// TwinCAT 3 PLC project sample_delivery
// ProgramVersion: 3.1.4023.0
// libraries:
//   lcls-twincat-sample-delivery, * (SLAC)
//   Tc2_Standard, * (Beckhoff Automation GmbH)
//   Tc2_System, * (Beckhoff Automation GmbH)
//   Tc3_Module, * (Beckhoff Automation GmbH)
// project tree:
//   GVLs/ GVL_SDS.TcGVL
//   / PlcTask.TcTTO, SerialComm.TcTTO
//   POUs/ MAIN.TcPOU, SerialTxRx.TcPOU (not stored)
// real-time tasks:
//   TASK PlcTask: cycle T#10ms, priority 20, ADS port 350
//   TASK SerialComm: cycle T#10ms, priority 1, ADS port 351
// I/O:
//   DEVICE Device 1 (EtherCAT), AmsNetId 172.21.38.25.2.1
//     Term 1 (EK1200)
//     Box 17 (EP9128-0021) [EP9128-0021 8x EtherCAT junction]
//       Term 18 (EP9128-1021) [EP9128-1021 8x EtherCAT junction - Dev A]
//         Box 20 (EP9128-0021)
//       Term 24 (EP9128-2021) [EP9128-2021 8x EtherCAT junction - Dev B]
//     ALI (EP1111) [EP1111-0000 ID-Switch]
//     ALI_X (EP7041-0002)
//     ALI_Y (EP7041-0002)
//     ALI_Z (EP7041-0002)
//     ALI_X_ENC (EP5101-0011)
//     ALI_Gauges (EP3174-0002)
//     ALI_PropValve (EP7041-0002)
//     ALI_Y_ENC (EP5101-0011)
//     ALI_DIO (EP2338-0001)
//     M3 Selector A (EP1111)
//     M3 Selector A Digital IO (EP2338-1001)
//     M3 Selector A Serial IO (EP6002-0002)
//     M3 Selector B (EP1111)
//     M3 Selector B Digital IO (EP2338-1001)
//     M3 Selector B Serial IO (EP6002-0002)
//     PCM A (EP1111) [EP1111-0000 ID-Switch]
//     PCM A (EP4374-0002)
//     PCM A (EP3174-0002)
//     PCM A (EP6002-0002)
//     PCM B (EP1111)
//     PCM B (EP4374-0002)
//     PCM B (EP3174-0002)
//     PCM B (EP6002-0002)
//     Gas_Mani (EP1111)
//     Gas_Mani_NeedleValve (EP4374-0002)
//     Gas_Mani_ValveCtrl (EP2338-0001)
//     Gas_Mani_ValveRbk (EP2338-0001)
//     M3 Selector C (EP1111)
//     M3 Selector C Digital IO (EP2338-1001)
//     M3 Selector C Serial IO (EP6002-0002)
//     M3 Selector D (EP1111)
//     M3 Selector D Digital IO (EP2338-1001)
//     M3 Selector D Serial IO (EP6002-0002)
//     PCM C (EP1111)
//     PCM C (EP4374-0002)
//     PCM C (EP3174-0002)
//     PCM C (EP6002-0002)
//     PCM D (EP1111)
//     PCM D (EP4374-0002)
//     PCM D (EP3174-0002)
//     PCM D (EP6002-0002)
//     Bronkhorst MFM A
//     Bronkhorst MFM B
//     Bronkhorst MFM C
//     Bronkhorst MFM D
//     Solenoid Pair A (EP1111)
//     Solenoid Pair A Digital IO (EP2338-0001)
// variable links:
//   sample-delivery Instance <-> Device 1 (EtherCAT)/Bronkhorst MFM B
//     PlcTask Inputs/GVL_SDS.BronkhorstB.stMFM.i_rFlow <-> TxPDO Map/fMeasure
//     PlcTask Outputs/GVL_SDS.BronkhorstB.stMFM.q_rSetpoint <-> RxPDO Map/fSetpoint
//   sample-delivery Instance <-> Device 1 (EtherCAT)/Gas_Mani_ValveCtrl (EP2338-0001)
//     PlcTask Outputs/GVL_SDS.GasMan.stValve[{1..7}].qxDO <-> Channel {9..15}/Output  (7 links)
//   sample-delivery Instance <-> Device 1 (EtherCAT)/Gas_Mani_ValveRbk (EP2338-0001)
//     PlcTask Inputs/GVL_SDS.GasMan.stValve[{1..7}].ixOPN <-> Channel {1..7}/Input  (7 links)
//   sample-delivery Instance <-> Device 1 (EtherCAT)/M3 Selector A Digital IO (EP2338-1001)
//     PlcTask Outputs/GVL_SDS.M3SelectorA.stShaker01.q_xPwrDO <-> Channel 9/Output
//     PlcTask Outputs/GVL_SDS.M3SelectorA.stShaker02.q_xPwrDO <-> Channel 10/Output
//     PlcTask Outputs/GVL_SDS.M3SelectorA.stShaker03.q_xPwrDO <-> Channel 11/Output
//     PlcTask Outputs/GVL_SDS.M3SelectorA.stShaker04.q_xPwrDO <-> Channel 12/Output
//   sample-delivery Instance <-> Device 1 (EtherCAT)/M3 Selector A Serial IO (EP6002-0002)
//     SerialComm Inputs/GVL_SDS.M3SelectorA.stSensSerial.stComIn/Status <-> COM TxPDO-Map Inputs Channel 1/Status
//     SerialComm Inputs/GVL_SDS.M3SelectorA.stViciSerial.stComIn/Status <-> COM TxPDO-Map Inputs Channel 2/Status
//   sample-delivery Instance <-> Device 1 (EtherCAT)/M3 Selector B Digital IO (EP2338-1001)
//     PlcTask Outputs/GVL_SDS.M3SelectorB.stShaker01.q_xPwrDO <-> Channel 9/Output
//     PlcTask Outputs/GVL_SDS.M3SelectorB.stShaker02.q_xPwrDO <-> Channel 10/Output
//     PlcTask Outputs/GVL_SDS.M3SelectorB.stShaker03.q_xPwrDO <-> Channel 11/Output
//     PlcTask Outputs/GVL_SDS.M3SelectorB.stShaker04.q_xPwrDO <-> Channel 12/Output
//   sample-delivery Instance <-> Device 1 (EtherCAT)/M3 Selector B Serial IO (EP6002-0002)
//     SerialComm Inputs/GVL_SDS.M3SelectorB.stSensSerial.stComIn/Status <-> COM TxPDO-Map Inputs Channel 1/Status
//     SerialComm Inputs/GVL_SDS.M3SelectorB.stViciSerial.stComIn/Status <-> COM TxPDO-Map Inputs Channel 2/Status
//   sample-delivery Instance <-> Device 1 (EtherCAT)/M3 Selector C Digital IO (EP2338-1001)
//     PlcTask Outputs/GVL_SDS.M3SelectorC.stShaker01.q_xPwrDO <-> Channel 9/Output
//     PlcTask Outputs/GVL_SDS.M3SelectorC.stShaker02.q_xPwrDO <-> Channel 10/Output
//     PlcTask Outputs/GVL_SDS.M3SelectorC.stShaker03.q_xPwrDO <-> Channel 11/Output
//     PlcTask Outputs/GVL_SDS.M3SelectorC.stShaker04.q_xPwrDO <-> Channel 12/Output
//   sample-delivery Instance <-> Device 1 (EtherCAT)/M3 Selector C Serial IO (EP6002-0002)
//     SerialComm Inputs/GVL_SDS.M3SelectorC.stSensSerial.stComIn/Status <-> COM TxPDO-Map Inputs Channel 1/Status
//     SerialComm Inputs/GVL_SDS.M3SelectorC.stViciSerial.stComIn/Status <-> COM TxPDO-Map Inputs Channel 2/Status
//   sample-delivery Instance <-> Device 1 (EtherCAT)/M3 Selector D Digital IO (EP2338-1001)
//     PlcTask Outputs/GVL_SDS.M3SelectorD.stShaker01.q_xPwrDO <-> Channel 9/Output
//     PlcTask Outputs/GVL_SDS.M3SelectorD.stShaker02.q_xPwrDO <-> Channel 10/Output
//     PlcTask Outputs/GVL_SDS.M3SelectorD.stShaker03.q_xPwrDO <-> Channel 11/Output
//     PlcTask Outputs/GVL_SDS.M3SelectorD.stShaker04.q_xPwrDO <-> Channel 12/Output
//   sample-delivery Instance <-> Device 1 (EtherCAT)/M3 Selector D Serial IO (EP6002-0002)
//     SerialComm Inputs/GVL_SDS.M3SelectorD.stSensSerial.stComIn/Status <-> COM TxPDO-Map Inputs Channel 1/Status
//     SerialComm Inputs/GVL_SDS.M3SelectorD.stViciSerial.stComIn/Status <-> COM TxPDO-Map Inputs Channel 2/Status
//   sample-delivery Instance <-> Device 1 (EtherCAT)/PCM A (EP1111)
//     PlcTask Inputs/GVL_SDS.PCMA.stBaseIO.i_SyncUnitWC <-> WcState/WcState
//   sample-delivery Instance <-> Device 1 (EtherCAT)/PCM A (EP4374-0002)
//     PlcTask Inputs/GVL_SDS.PCMA.stPropAir1.i_iPressRB <-> AI Inputs Channel 1/Value
//     PlcTask Inputs/GVL_SDS.PCMA.stPropAir2.i_iPressRB <-> AI Inputs Channel 2/Value
//     PlcTask Outputs/GVL_SDS.PCMA.stPropAir1.q_iPressCt <-> AO Outputs Channel 3/Analog output
//     PlcTask Outputs/GVL_SDS.PCMA.stPropAir2.q_iPressCt <-> AO Outputs Channel 4/Analog output
//   sample-delivery Instance <-> Device 1 (EtherCAT)/PCM A (EP6002-0002)
//     SerialComm Inputs/GVL_SDS.PCMA.stSerial1.stComIn/D[0] <-> COM TxPDO-Map Inputs Channel 1/Data In 0
//     SerialComm Inputs/GVL_SDS.PCMA.stSerial1.stComIn/D[10] <-> COM TxPDO-Map Inputs Channel 1/Data In 10
//     SerialComm Inputs/GVL_SDS.PCMA.stSerial1.stComIn/D[11] <-> COM TxPDO-Map Inputs Channel 1/Data In 11
//     SerialComm Inputs/GVL_SDS.PCMA.stSerial1.stComIn/D[12] <-> COM TxPDO-Map Inputs Channel 1/Data In 12
//     SerialComm Inputs/GVL_SDS.PCMA.stSerial1.stComIn/D[13] <-> COM TxPDO-Map Inputs Channel 1/Data In 13
//     SerialComm Inputs/GVL_SDS.PCMA.stSerial1.stComIn/D[14] <-> COM TxPDO-Map Inputs Channel 1/Data In 14
//     SerialComm Inputs/GVL_SDS.PCMA.stSerial1.stComIn/D[15] <-> COM TxPDO-Map Inputs Channel 1/Data In 15
//     SerialComm Inputs/GVL_SDS.PCMA.stSerial1.stComIn/D[16] <-> COM TxPDO-Map Inputs Channel 1/Data In 16
//     SerialComm Inputs/GVL_SDS.PCMA.stSerial1.stComIn/D[17] <-> COM TxPDO-Map Inputs Channel 1/Data In 17
//     SerialComm Inputs/GVL_SDS.PCMA.stSerial1.stComIn/D[18] <-> COM TxPDO-Map Inputs Channel 1/Data In 18
//     SerialComm Inputs/GVL_SDS.PCMA.stSerial1.stComIn/D[19] <-> COM TxPDO-Map Inputs Channel 1/Data In 19
//     SerialComm Inputs/GVL_SDS.PCMA.stSerial1.stComIn/D[1] <-> COM TxPDO-Map Inputs Channel 1/Data In 1
//     SerialComm Inputs/GVL_SDS.PCMA.stSerial1.stComIn/D[20] <-> COM TxPDO-Map Inputs Channel 1/Data In 20
//     SerialComm Inputs/GVL_SDS.PCMA.stSerial1.stComIn/D[21] <-> COM TxPDO-Map Inputs Channel 1/Data In 21
//     SerialComm Inputs/GVL_SDS.PCMA.stSerial1.stComIn/D[2] <-> COM TxPDO-Map Inputs Channel 1/Data In 2
//     SerialComm Inputs/GVL_SDS.PCMA.stSerial1.stComIn/D[3] <-> COM TxPDO-Map Inputs Channel 1/Data In 3
//     SerialComm Inputs/GVL_SDS.PCMA.stSerial1.stComIn/D[4] <-> COM TxPDO-Map Inputs Channel 1/Data In 4
//     SerialComm Inputs/GVL_SDS.PCMA.stSerial1.stComIn/D[5] <-> COM TxPDO-Map Inputs Channel 1/Data In 5
//     SerialComm Inputs/GVL_SDS.PCMA.stSerial1.stComIn/D[6] <-> COM TxPDO-Map Inputs Channel 1/Data In 6
//     SerialComm Inputs/GVL_SDS.PCMA.stSerial1.stComIn/D[7] <-> COM TxPDO-Map Inputs Channel 1/Data In 7
//     SerialComm Inputs/GVL_SDS.PCMA.stSerial1.stComIn/D[8] <-> COM TxPDO-Map Inputs Channel 1/Data In 8
//     SerialComm Inputs/GVL_SDS.PCMA.stSerial1.stComIn/D[9] <-> COM TxPDO-Map Inputs Channel 1/Data In 9
//     SerialComm Inputs/GVL_SDS.PCMA.stSerial2.stComIn/D[0] <-> COM TxPDO-Map Inputs Channel 2/Data In 0
//     SerialComm Inputs/GVL_SDS.PCMA.stSerial2.stComIn/D[10] <-> COM TxPDO-Map Inputs Channel 2/Data In 10
//     SerialComm Inputs/GVL_SDS.PCMA.stSerial2.stComIn/D[11] <-> COM TxPDO-Map Inputs Channel 2/Data In 11
//     SerialComm Inputs/GVL_SDS.PCMA.stSerial2.stComIn/D[12] <-> COM TxPDO-Map Inputs Channel 2/Data In 12
//     SerialComm Inputs/GVL_SDS.PCMA.stSerial2.stComIn/D[13] <-> COM TxPDO-Map Inputs Channel 2/Data In 13
//     SerialComm Inputs/GVL_SDS.PCMA.stSerial2.stComIn/D[14] <-> COM TxPDO-Map Inputs Channel 2/Data In 14
//     SerialComm Inputs/GVL_SDS.PCMA.stSerial2.stComIn/D[15] <-> COM TxPDO-Map Inputs Channel 2/Data In 15
//     SerialComm Inputs/GVL_SDS.PCMA.stSerial2.stComIn/D[16] <-> COM TxPDO-Map Inputs Channel 2/Data In 16
//     SerialComm Inputs/GVL_SDS.PCMA.stSerial2.stComIn/D[17] <-> COM TxPDO-Map Inputs Channel 2/Data In 17
//     SerialComm Inputs/GVL_SDS.PCMA.stSerial2.stComIn/D[18] <-> COM TxPDO-Map Inputs Channel 2/Data In 18
//     SerialComm Inputs/GVL_SDS.PCMA.stSerial2.stComIn/D[19] <-> COM TxPDO-Map Inputs Channel 2/Data In 19
//     SerialComm Inputs/GVL_SDS.PCMA.stSerial2.stComIn/D[1] <-> COM TxPDO-Map Inputs Channel 2/Data In 1
//     SerialComm Inputs/GVL_SDS.PCMA.stSerial2.stComIn/D[20] <-> COM TxPDO-Map Inputs Channel 2/Data In 20
//     SerialComm Inputs/GVL_SDS.PCMA.stSerial2.stComIn/D[21] <-> COM TxPDO-Map Inputs Channel 2/Data In 21
//     SerialComm Inputs/GVL_SDS.PCMA.stSerial2.stComIn/D[2] <-> COM TxPDO-Map Inputs Channel 2/Data In 2
//     SerialComm Inputs/GVL_SDS.PCMA.stSerial2.stComIn/D[3] <-> COM TxPDO-Map Inputs Channel 2/Data In 3
//     SerialComm Inputs/GVL_SDS.PCMA.stSerial2.stComIn/D[4] <-> COM TxPDO-Map Inputs Channel 2/Data In 4
//     SerialComm Inputs/GVL_SDS.PCMA.stSerial2.stComIn/D[5] <-> COM TxPDO-Map Inputs Channel 2/Data In 5
//     SerialComm Inputs/GVL_SDS.PCMA.stSerial2.stComIn/D[6] <-> COM TxPDO-Map Inputs Channel 2/Data In 6
//     SerialComm Inputs/GVL_SDS.PCMA.stSerial2.stComIn/D[7] <-> COM TxPDO-Map Inputs Channel 2/Data In 7
//     SerialComm Inputs/GVL_SDS.PCMA.stSerial2.stComIn/D[8] <-> COM TxPDO-Map Inputs Channel 2/Data In 8
//     SerialComm Inputs/GVL_SDS.PCMA.stSerial2.stComIn/D[9] <-> COM TxPDO-Map Inputs Channel 2/Data In 9
//     SerialComm Inputs/GVL_SDS.PCMA.stSerial1.stComIn/Status <-> COM TxPDO-Map Inputs Channel 1/Status
//     SerialComm Inputs/GVL_SDS.PCMA.stSerial2.stComIn/Status <-> COM TxPDO-Map Inputs Channel 2/Status
//     SerialComm Outputs/GVL_SDS.PCMA.stSerial1.stComOut/Ctrl <-> COM RxPDO-Map Outputs Channel 1/Ctrl
//     SerialComm Outputs/GVL_SDS.PCMA.stSerial2.stComOut/Ctrl <-> COM RxPDO-Map Outputs Channel 2/Ctrl
//     SerialComm Outputs/GVL_SDS.PCMA.stSerial1.stComOut/D[0] <-> COM RxPDO-Map Outputs Channel 1/Data Out 0
//     SerialComm Outputs/GVL_SDS.PCMA.stSerial1.stComOut/D[10] <-> COM RxPDO-Map Outputs Channel 1/Data Out 10
//     SerialComm Outputs/GVL_SDS.PCMA.stSerial1.stComOut/D[11] <-> COM RxPDO-Map Outputs Channel 1/Data Out 11
//     SerialComm Outputs/GVL_SDS.PCMA.stSerial1.stComOut/D[12] <-> COM RxPDO-Map Outputs Channel 1/Data Out 12
//     SerialComm Outputs/GVL_SDS.PCMA.stSerial1.stComOut/D[13] <-> COM RxPDO-Map Outputs Channel 1/Data Out 13
//     SerialComm Outputs/GVL_SDS.PCMA.stSerial1.stComOut/D[14] <-> COM RxPDO-Map Outputs Channel 1/Data Out 14
//     SerialComm Outputs/GVL_SDS.PCMA.stSerial1.stComOut/D[15] <-> COM RxPDO-Map Outputs Channel 1/Data Out 15
//     SerialComm Outputs/GVL_SDS.PCMA.stSerial1.stComOut/D[16] <-> COM RxPDO-Map Outputs Channel 1/Data Out 16
//     SerialComm Outputs/GVL_SDS.PCMA.stSerial1.stComOut/D[17] <-> COM RxPDO-Map Outputs Channel 1/Data Out 17
//     SerialComm Outputs/GVL_SDS.PCMA.stSerial1.stComOut/D[18] <-> COM RxPDO-Map Outputs Channel 1/Data Out 18
//     SerialComm Outputs/GVL_SDS.PCMA.stSerial1.stComOut/D[19] <-> COM RxPDO-Map Outputs Channel 1/Data Out 19
//     SerialComm Outputs/GVL_SDS.PCMA.stSerial1.stComOut/D[1] <-> COM RxPDO-Map Outputs Channel 1/Data Out 1
//     SerialComm Outputs/GVL_SDS.PCMA.stSerial1.stComOut/D[20] <-> COM RxPDO-Map Outputs Channel 1/Data Out 20
//     SerialComm Outputs/GVL_SDS.PCMA.stSerial1.stComOut/D[21] <-> COM RxPDO-Map Outputs Channel 1/Data Out 21
//     SerialComm Outputs/GVL_SDS.PCMA.stSerial1.stComOut/D[2] <-> COM RxPDO-Map Outputs Channel 1/Data Out 2
//     SerialComm Outputs/GVL_SDS.PCMA.stSerial1.stComOut/D[3] <-> COM RxPDO-Map Outputs Channel 1/Data Out 3
//     SerialComm Outputs/GVL_SDS.PCMA.stSerial1.stComOut/D[4] <-> COM RxPDO-Map Outputs Channel 1/Data Out 4
//     SerialComm Outputs/GVL_SDS.PCMA.stSerial1.stComOut/D[5] <-> COM RxPDO-Map Outputs Channel 1/Data Out 5
//     SerialComm Outputs/GVL_SDS.PCMA.stSerial1.stComOut/D[6] <-> COM RxPDO-Map Outputs Channel 1/Data Out 6
//     SerialComm Outputs/GVL_SDS.PCMA.stSerial1.stComOut/D[7] <-> COM RxPDO-Map Outputs Channel 1/Data Out 7
//     SerialComm Outputs/GVL_SDS.PCMA.stSerial1.stComOut/D[8] <-> COM RxPDO-Map Outputs Channel 1/Data Out 8
//     SerialComm Outputs/GVL_SDS.PCMA.stSerial1.stComOut/D[9] <-> COM RxPDO-Map Outputs Channel 1/Data Out 9
//     SerialComm Outputs/GVL_SDS.PCMA.stSerial2.stComOut/D[0] <-> COM RxPDO-Map Outputs Channel 2/Data Out 0
//     SerialComm Outputs/GVL_SDS.PCMA.stSerial2.stComOut/D[10] <-> COM RxPDO-Map Outputs Channel 2/Data Out 10
//     SerialComm Outputs/GVL_SDS.PCMA.stSerial2.stComOut/D[11] <-> COM RxPDO-Map Outputs Channel 2/Data Out 11
//     SerialComm Outputs/GVL_SDS.PCMA.stSerial2.stComOut/D[12] <-> COM RxPDO-Map Outputs Channel 2/Data Out 12
//     SerialComm Outputs/GVL_SDS.PCMA.stSerial2.stComOut/D[13] <-> COM RxPDO-Map Outputs Channel 2/Data Out 13
//     SerialComm Outputs/GVL_SDS.PCMA.stSerial2.stComOut/D[14] <-> COM RxPDO-Map Outputs Channel 2/Data Out 14
//     SerialComm Outputs/GVL_SDS.PCMA.stSerial2.stComOut/D[15] <-> COM RxPDO-Map Outputs Channel 2/Data Out 15
//     SerialComm Outputs/GVL_SDS.PCMA.stSerial2.stComOut/D[16] <-> COM RxPDO-Map Outputs Channel 2/Data Out 16
//     SerialComm Outputs/GVL_SDS.PCMA.stSerial2.stComOut/D[17] <-> COM RxPDO-Map Outputs Channel 2/Data Out 17
//     SerialComm Outputs/GVL_SDS.PCMA.stSerial2.stComOut/D[18] <-> COM RxPDO-Map Outputs Channel 2/Data Out 18
//     SerialComm Outputs/GVL_SDS.PCMA.stSerial2.stComOut/D[19] <-> COM RxPDO-Map Outputs Channel 2/Data Out 19
//     SerialComm Outputs/GVL_SDS.PCMA.stSerial2.stComOut/D[1] <-> COM RxPDO-Map Outputs Channel 2/Data Out 1
//     SerialComm Outputs/GVL_SDS.PCMA.stSerial2.stComOut/D[20] <-> COM RxPDO-Map Outputs Channel 2/Data Out 20
//     SerialComm Outputs/GVL_SDS.PCMA.stSerial2.stComOut/D[21] <-> COM RxPDO-Map Outputs Channel 2/Data Out 21
//     SerialComm Outputs/GVL_SDS.PCMA.stSerial2.stComOut/D[2] <-> COM RxPDO-Map Outputs Channel 2/Data Out 2
//     SerialComm Outputs/GVL_SDS.PCMA.stSerial2.stComOut/D[3] <-> COM RxPDO-Map Outputs Channel 2/Data Out 3
//     SerialComm Outputs/GVL_SDS.PCMA.stSerial2.stComOut/D[4] <-> COM RxPDO-Map Outputs Channel 2/Data Out 4
//     SerialComm Outputs/GVL_SDS.PCMA.stSerial2.stComOut/D[5] <-> COM RxPDO-Map Outputs Channel 2/Data Out 5
//     SerialComm Outputs/GVL_SDS.PCMA.stSerial2.stComOut/D[6] <-> COM RxPDO-Map Outputs Channel 2/Data Out 6
//     SerialComm Outputs/GVL_SDS.PCMA.stSerial2.stComOut/D[7] <-> COM RxPDO-Map Outputs Channel 2/Data Out 7
//     SerialComm Outputs/GVL_SDS.PCMA.stSerial2.stComOut/D[8] <-> COM RxPDO-Map Outputs Channel 2/Data Out 8
//     SerialComm Outputs/GVL_SDS.PCMA.stSerial2.stComOut/D[9] <-> COM RxPDO-Map Outputs Channel 2/Data Out 9
//   sample-delivery Instance <-> Device 1 (EtherCAT)/PCM B (EP1111)
//     PlcTask Inputs/GVL_SDS.PCMB.stBaseIO.i_SyncUnitWC <-> WcState/WcState
//   sample-delivery Instance <-> Device 1 (EtherCAT)/PCM B (EP4374-0002)
//     PlcTask Inputs/GVL_SDS.PCMB.stPropAir1.i_iPressRB <-> AI Inputs Channel 1/Value
//     PlcTask Inputs/GVL_SDS.PCMB.stPropAir2.i_iPressRB <-> AI Inputs Channel 2/Value
//     PlcTask Outputs/GVL_SDS.PCMB.stPropAir1.q_iPressCt <-> AO Outputs Channel 3/Analog output
//     PlcTask Outputs/GVL_SDS.PCMB.stPropAir2.q_iPressCt <-> AO Outputs Channel 4/Analog output
//   sample-delivery Instance <-> Device 1 (EtherCAT)/PCM B (EP6002-0002)
//     SerialComm Inputs/GVL_SDS.PCMB.stSerial1.stComIn/Status <-> COM TxPDO-Map Inputs Channel 1/Status
//     SerialComm Inputs/GVL_SDS.PCMB.stSerial2.stComIn/Status <-> COM TxPDO-Map Inputs Channel 2/Status
//     SerialComm Outputs/GVL_SDS.PCMB.stSerial1.stComOut/Ctrl <-> COM RxPDO-Map Outputs Channel 1/Ctrl
//     SerialComm Outputs/GVL_SDS.PCMB.stSerial2.stComOut/Ctrl <-> COM RxPDO-Map Outputs Channel 2/Ctrl
//   sample-delivery Instance <-> Device 1 (EtherCAT)/PCM C (EP1111)
//     PlcTask Inputs/GVL_SDS.PCMC.stBaseIO.i_SyncUnitWC <-> WcState/WcState
//   sample-delivery Instance <-> Device 1 (EtherCAT)/PCM C (EP4374-0002)
//     PlcTask Inputs/GVL_SDS.PCMC.stPropAir1.i_iPressRB <-> AI Inputs Channel 1/Value
//     PlcTask Inputs/GVL_SDS.PCMC.stPropAir2.i_iPressRB <-> AI Inputs Channel 2/Value
//     PlcTask Outputs/GVL_SDS.PCMC.stPropAir1.q_iPressCt <-> AO Outputs Channel 3/Analog output
//     PlcTask Outputs/GVL_SDS.PCMC.stPropAir2.q_iPressCt <-> AO Outputs Channel 4/Analog output
//   sample-delivery Instance <-> Device 1 (EtherCAT)/PCM C (EP6002-0002)
//     SerialComm Inputs/GVL_SDS.PCMC.stSerial1.stComIn/Status <-> COM TxPDO-Map Inputs Channel 1/Status
//     SerialComm Inputs/GVL_SDS.PCMC.stSerial2.stComIn/Status <-> COM TxPDO-Map Inputs Channel 2/Status
//     SerialComm Outputs/GVL_SDS.PCMC.stSerial1.stComOut/Ctrl <-> COM RxPDO-Map Outputs Channel 1/Ctrl
//     SerialComm Outputs/GVL_SDS.PCMC.stSerial2.stComOut/Ctrl <-> COM RxPDO-Map Outputs Channel 2/Ctrl
//   sample-delivery Instance <-> Device 1 (EtherCAT)/PCM D (EP1111)
//     PlcTask Inputs/GVL_SDS.PCMD.stBaseIO.i_SyncUnitWC <-> WcState/WcState
//   sample-delivery Instance <-> Device 1 (EtherCAT)/PCM D (EP4374-0002)
//     PlcTask Inputs/GVL_SDS.PCMD.stPropAir1.i_iPressRB <-> AI Inputs Channel 1/Value
//     PlcTask Inputs/GVL_SDS.PCMD.stPropAir2.i_iPressRB <-> AI Inputs Channel 2/Value
//     PlcTask Outputs/GVL_SDS.PCMD.stPropAir1.q_iPressCt <-> AO Outputs Channel 3/Analog output
//     PlcTask Outputs/GVL_SDS.PCMD.stPropAir2.q_iPressCt <-> AO Outputs Channel 4/Analog output
//   sample-delivery Instance <-> Device 1 (EtherCAT)/PCM D (EP6002-0002)
//     SerialComm Inputs/GVL_SDS.PCMD.stSerial1.stComIn/Status <-> COM TxPDO-Map Inputs Channel 1/Status
//     SerialComm Inputs/GVL_SDS.PCMD.stSerial2.stComIn/Status <-> COM TxPDO-Map Inputs Channel 2/Status
//     SerialComm Outputs/GVL_SDS.PCMD.stSerial1.stComOut/Ctrl <-> COM RxPDO-Map Outputs Channel 1/Ctrl
//     SerialComm Outputs/GVL_SDS.PCMD.stSerial2.stComOut/Ctrl <-> COM RxPDO-Map Outputs Channel 2/Ctrl
//   sample-delivery Instance <-> Device 1 (EtherCAT)/Solenoid Pair A Digital IO (EP2338-0001)
//     PlcTask Outputs/GVL_SDS.SolenoidPairA.q_xDO1 <-> Channel 9/Output
//     PlcTask Outputs/GVL_SDS.SolenoidPairA.q_xDO2 <-> Channel 10/Output

CONFIGURATION sample_delivery
    RESOURCE PLC ON TwinCAT3
        TASK PlcTask(INTERVAL := T#10ms, PRIORITY := 20);
        TASK SerialComm(INTERVAL := T#10ms, PRIORITY := 1);
        PROGRAM MAIN WITH PlcTask : MAIN;
        PROGRAM SerialTxRx WITH SerialComm : SerialTxRx;
    END_RESOURCE
END_CONFIGURATION

// ---- GVLs/GVL_SDS.TcGVL
VAR_GLOBAL
	
// TODO: FIX Linking for Devices will be deployed
//  Working: Bronkhorst MFM B
{attribute 'pytmc' := 'pv: XCS:SDS:SEL:A'}
{attribute 'TcLinkTo' := '.stSensSerial.stComIn.Status := TIIB[M3 Selector A Serial IO (EP6002-0002)]^COM TxPDO-Map Inputs Channel 1^Status;
                          .stViciSerial.stComIn.Status := TIIB[M3 Selector A Serial IO (EP6002-0002)]^COM TxPDO-Map Inputs Channel 2^Status;
                          .stSensSerial.stComOut.Ctrl := TIID^MAIN (EtherCAT)^M3 Selector A Serial IO (EP6002-0002)^COM RxPDO-Map Outputs Channel 1^Ctrl;
                          .stViciSerial.stComOut.Ctrl := TIID^MAIN (EtherCAT)^M3 Selector A Serial IO (EP6002-0002)^COM RxPDO-Map Outputs Channel 2^Ctrl;
                          .stShaker01.q_xPwrDO := TIIB[M3 Selector A Digital IO (EP2338-1001)]^Channel 9^Output;
                          .stShaker02.q_xPwrDO := TIIB[M3 Selector A Digital IO (EP2338-1001)]^Channel 10^Output;
                          .stShaker03.q_xPwrDO := TIIB[M3 Selector A Digital IO (EP2338-1001)]^Channel 11^Output;
                          .stShaker04.q_xPwrDO := TIIB[M3 Selector A Digital IO (EP2338-1001)]^Channel 12^Output;
                          .stBaseIO.i_SyncUnitWC := TIID^MAIN (EtherCAT)^M3 Selector A (EP1111)^WcState^WcState;
						  .
'}
M3SelectorA : FB_SelectorM3;

{attribute 'pytmc' := 'pv: XCS:SDS:SEL:B'}
{attribute 'TcLinkTo' := '.stSensSerial.stComIn.Status := TIIB[M3 Selector B Serial IO (EP6002-0002)]^COM TxPDO-Map Inputs Channel 1^Status;
                          .stViciSerial.stComIn.Status := TIIB[M3 Selector B Serial IO (EP6002-0002)]^COM TxPDO-Map Inputs Channel 2^Status;
                          .stSensSerial.stComOut.Ctrl := TIID^MAIN (EtherCAT)^M3 Selector B Serial IO (EP6002-0002)^COM RxPDO-Map Outputs Channel 1^Ctrl;
                          .stViciSerial.stComOut.Ctrl := TIID^MAIN (EtherCAT)^M3 Selector B Serial IO (EP6002-0002)^COM RxPDO-Map Outputs Channel 2^Ctrl;
                          .stShaker01.q_xPwrDO := TIIB[M3 Selector B Digital IO (EP2338-1001)]^Channel 9^Output;
                          .stShaker02.q_xPwrDO := TIIB[M3 Selector B Digital IO (EP2338-1001)]^Channel 10^Output;
                          .stShaker03.q_xPwrDO := TIIB[M3 Selector B Digital IO (EP2338-1001)]^Channel 11^Output;
                          .stShaker04.q_xPwrDO := TIIB[M3 Selector B Digital IO (EP2338-1001)]^Channel 12^Output;
                          .stBaseIO.i_SyncUnitWC := TIID^MAIN (EtherCAT)^M3 Selector B (EP1111)^WcState^WcState
'}
M3SelectorB : FB_SelectorM3;

{attribute 'pytmc' := 'pv: XCS:SDS:SEL:C'}
{attribute 'TcLinkTo' := '.stSensSerial.stComIn.Status := TIIB[M3 Selector C Serial IO (EP6002-0002)]^COM TxPDO-Map Inputs Channel 1^Status;
                          .stViciSerial.stComIn.Status := TIIB[M3 Selector C Serial IO (EP6002-0002)]^COM TxPDO-Map Inputs Channel 2^Status;
                          .stSensSerial.stComOut.Ctrl := TIID^MAIN (EtherCAT)^M3 Selector C Serial IO (EP6002-0002)^COM RxPDO-Map Outputs Channel 1^Ctrl;
                          .stViciSerial.stComOut.Ctrl := TIID^MAIN (EtherCAT)^M3 Selector C Serial IO (EP6002-0002)^COM RxPDO-Map Outputs Channel 2^Ctrl;
                          .stShaker01.q_xPwrDO := TIIB[M3 Selector C Digital IO (EP2338-1001)]^Channel 9^Output;
                          .stShaker02.q_xPwrDO := TIIB[M3 Selector C Digital IO (EP2338-1001)]^Channel 10^Output;
                          .stShaker03.q_xPwrDO := TIIB[M3 Selector C Digital IO (EP2338-1001)]^Channel 11^Output;
                          .stShaker04.q_xPwrDO := TIIB[M3 Selector C Digital IO (EP2338-1001)]^Channel 12^Output;
                          .stBaseIO.i_SyncUnitWC := TIID^MAIN (EtherCAT)^M3 Selector C (EP1111)^WcState^WcState
'}
M3SelectorC : FB_SelectorM3;

{attribute 'pytmc' := 'pv: XCS:SDS:SEL:D'}
{attribute 'TcLinkTo' := '.stSensSerial.stComIn.Status := TIIB[M3 Selector D Serial IO (EP6002-0002)]^COM TxPDO-Map Inputs Channel 1^Status;
                          .stViciSerial.stComIn.Status := TIIB[M3 Selector D Serial IO (EP6002-0002)]^COM TxPDO-Map Inputs Channel 2^Status;
                          .stSensSerial.stComOut.Ctrl := TIID^MAIN (EtherCAT)^M3 Selector D Serial IO (EP6002-0002)^COM RxPDO-Map Outputs Channel 1^Ctrl;
                          .stViciSerial.stComOut.Ctrl := TIID^MAIN (EtherCAT)^M3 Selector D Serial IO (EP6002-0002)^COM RxPDO-Map Outputs Channel 2^Ctrl;
                          .stShaker01.q_xPwrDO := TIIB[M3 Selector D Digital IO (EP2338-1001)]^Channel 9^Output;
                          .stShaker02.q_xPwrDO := TIIB[M3 Selector D Digital IO (EP2338-1001)]^Channel 10^Output;
                          .stShaker03.q_xPwrDO := TIIB[M3 Selector D Digital IO (EP2338-1001)]^Channel 11^Output;
                          .stShaker04.q_xPwrDO := TIIB[M3 Selector D Digital IO (EP2338-1001)]^Channel 12^Output;
                          .stBaseIO.i_SyncUnitWC := TIID^MAIN (EtherCAT)^M3 Selector D (EP1111)^WcState^WcState
'}
M3SelectorD : FB_SelectorM3;

{attribute 'pytmc' := 'pv: XCS:SDS:PCM:A'}
{attribute 'TcLinkTo' := '.stPropAir1.i_iPressRB 		:= TIIB[PCM A (EP4374-0002)]^AI Inputs Channel 1^Value;
                          .stPropAir2.i_iPressRB 		:= TIIB[PCM A (EP4374-0002)]^AI Inputs Channel 2^Value;
                          .stPropAir1.q_iPressCt 		:= TIIB[PCM A (EP4374-0002)]^AO Outputs Channel 3^Analog output;
                          .stPropAir2.q_iPressCt 		:= TIIB[PCM A (EP4374-0002)]^AO Outputs Channel 4^Analog output;
                          .stSerial1.stComIn.Status 	:= TIIB[PCM A (EP6002-0002)]^COM TxPDO-Map Inputs Channel 1^Status;
                          .stSerial2.stComIn.Status 	:= TIIB[PCM A (EP6002-0002)]^COM TxPDO-Map Inputs Channel 2^Status;
                          .stSerial1.stComOut.Ctrl 		:= TIIB[PCM A (EP6002-0002)]^COM RxPDO-Map Outputs Channel 1^Ctrl;
                          .stSerial2.stComOut.Ctrl 		:= TIIB[PCM A (EP6002-0002)]^COM RxPDO-Map Outputs Channel 2^Ctrl;
                          .stBaseIO.i_SyncUnitWC 		:= TIIB[PCM A (EP1111)]^WcState^WcState;
						  
						  .stSerial1.stComIn.D[0]  		:= TIIB[PCM A (EP6002-0002)]^COM TxPDO-Map Inputs Channel 1^Data In 0;
						  .stSerial1.stComIn.D[1]  		:= TIIB[PCM A (EP6002-0002)]^COM TxPDO-Map Inputs Channel 1^Data In 1;
						  .stSerial1.stComIn.D[2]  		:= TIIB[PCM A (EP6002-0002)]^COM TxPDO-Map Inputs Channel 1^Data In 2;
						  .stSerial1.stComIn.D[3]  		:= TIIB[PCM A (EP6002-0002)]^COM TxPDO-Map Inputs Channel 1^Data In 3;
						  .stSerial1.stComIn.D[4]  		:= TIIB[PCM A (EP6002-0002)]^COM TxPDO-Map Inputs Channel 1^Data In 4;
						  .stSerial1.stComIn.D[5]  		:= TIIB[PCM A (EP6002-0002)]^COM TxPDO-Map Inputs Channel 1^Data In 5;
						  .stSerial1.stComIn.D[6]  		:= TIIB[PCM A (EP6002-0002)]^COM TxPDO-Map Inputs Channel 1^Data In 6;
						  .stSerial1.stComIn.D[7]  		:= TIIB[PCM A (EP6002-0002)]^COM TxPDO-Map Inputs Channel 1^Data In 7;
						  .stSerial1.stComIn.D[8]  		:= TIIB[PCM A (EP6002-0002)]^COM TxPDO-Map Inputs Channel 1^Data In 8;
						  .stSerial1.stComIn.D[9]  		:= TIIB[PCM A (EP6002-0002)]^COM TxPDO-Map Inputs Channel 1^Data In 9;
						  .stSerial1.stComIn.D[10]  	:= TIIB[PCM A (EP6002-0002)]^COM TxPDO-Map Inputs Channel 1^Data In 10;
						  .stSerial1.stComIn.D[11]  	:= TIIB[PCM A (EP6002-0002)]^COM TxPDO-Map Inputs Channel 1^Data In 11;
						  .stSerial1.stComIn.D[12]  	:= TIIB[PCM A (EP6002-0002)]^COM TxPDO-Map Inputs Channel 1^Data In 12;
						  .stSerial1.stComIn.D[13]  	:= TIIB[PCM A (EP6002-0002)]^COM TxPDO-Map Inputs Channel 1^Data In 13;
						  .stSerial1.stComIn.D[14]  	:= TIIB[PCM A (EP6002-0002)]^COM TxPDO-Map Inputs Channel 1^Data In 14;
						  .stSerial1.stComIn.D[15]  	:= TIIB[PCM A (EP6002-0002)]^COM TxPDO-Map Inputs Channel 1^Data In 15;
						  .stSerial1.stComIn.D[16]  	:= TIIB[PCM A (EP6002-0002)]^COM TxPDO-Map Inputs Channel 1^Data In 16;
						  .stSerial1.stComIn.D[17]  	:= TIIB[PCM A (EP6002-0002)]^COM TxPDO-Map Inputs Channel 1^Data In 17;
						  .stSerial1.stComIn.D[18]  	:= TIIB[PCM A (EP6002-0002)]^COM TxPDO-Map Inputs Channel 1^Data In 18;
						  .stSerial1.stComIn.D[19]  	:= TIIB[PCM A (EP6002-0002)]^COM TxPDO-Map Inputs Channel 1^Data In 19;
						  .stSerial1.stComIn.D[20]  	:= TIIB[PCM A (EP6002-0002)]^COM TxPDO-Map Inputs Channel 1^Data In 20;
						  .stSerial1.stComIn.D[21]  	:= TIIB[PCM A (EP6002-0002)]^COM TxPDO-Map Inputs Channel 1^Data In 21;
						  
						  .stSerial2.stComIn.D[0]  		:= TIIB[PCM A (EP6002-0002)]^COM TxPDO-Map Inputs Channel 2^Data In 0;
						  .stSerial2.stComIn.D[1]  		:= TIIB[PCM A (EP6002-0002)]^COM TxPDO-Map Inputs Channel 2^Data In 1;
						  .stSerial2.stComIn.D[2]  		:= TIIB[PCM A (EP6002-0002)]^COM TxPDO-Map Inputs Channel 2^Data In 2;
						  .stSerial2.stComIn.D[3]  		:= TIIB[PCM A (EP6002-0002)]^COM TxPDO-Map Inputs Channel 2^Data In 3;
						  .stSerial2.stComIn.D[4]  		:= TIIB[PCM A (EP6002-0002)]^COM TxPDO-Map Inputs Channel 2^Data In 4;
						  .stSerial2.stComIn.D[5]  		:= TIIB[PCM A (EP6002-0002)]^COM TxPDO-Map Inputs Channel 2^Data In 5;
						  .stSerial2.stComIn.D[6]  		:= TIIB[PCM A (EP6002-0002)]^COM TxPDO-Map Inputs Channel 2^Data In 6;
						  .stSerial2.stComIn.D[7]  		:= TIIB[PCM A (EP6002-0002)]^COM TxPDO-Map Inputs Channel 2^Data In 7;
						  .stSerial2.stComIn.D[8]  		:= TIIB[PCM A (EP6002-0002)]^COM TxPDO-Map Inputs Channel 2^Data In 8;
						  .stSerial2.stComIn.D[9]  		:= TIIB[PCM A (EP6002-0002)]^COM TxPDO-Map Inputs Channel 2^Data In 9;
						  .stSerial2.stComIn.D[10]  	:= TIIB[PCM A (EP6002-0002)]^COM TxPDO-Map Inputs Channel 2^Data In 10;
						  .stSerial2.stComIn.D[11]  	:= TIIB[PCM A (EP6002-0002)]^COM TxPDO-Map Inputs Channel 2^Data In 11;
						  .stSerial2.stComIn.D[12]  	:= TIIB[PCM A (EP6002-0002)]^COM TxPDO-Map Inputs Channel 2^Data In 12;
						  .stSerial2.stComIn.D[13]  	:= TIIB[PCM A (EP6002-0002)]^COM TxPDO-Map Inputs Channel 2^Data In 13;
						  .stSerial2.stComIn.D[14]  	:= TIIB[PCM A (EP6002-0002)]^COM TxPDO-Map Inputs Channel 2^Data In 14;
						  .stSerial2.stComIn.D[15]  	:= TIIB[PCM A (EP6002-0002)]^COM TxPDO-Map Inputs Channel 2^Data In 15;
						  .stSerial2.stComIn.D[16]  	:= TIIB[PCM A (EP6002-0002)]^COM TxPDO-Map Inputs Channel 2^Data In 16;
						  .stSerial2.stComIn.D[17]  	:= TIIB[PCM A (EP6002-0002)]^COM TxPDO-Map Inputs Channel 2^Data In 17;
						  .stSerial2.stComIn.D[18]  	:= TIIB[PCM A (EP6002-0002)]^COM TxPDO-Map Inputs Channel 2^Data In 18;
						  .stSerial2.stComIn.D[19]  	:= TIIB[PCM A (EP6002-0002)]^COM TxPDO-Map Inputs Channel 2^Data In 19;
						  .stSerial2.stComIn.D[20]  	:= TIIB[PCM A (EP6002-0002)]^COM TxPDO-Map Inputs Channel 2^Data In 20;
						  .stSerial2.stComIn.D[21]  	:= TIIB[PCM A (EP6002-0002)]^COM TxPDO-Map Inputs Channel 2^Data In 21;
						  
						  .stSerial1.stComOut.D[0]  		:= TIIB[PCM A (EP6002-0002)]^COM RxPDO-Map Outputs Channel 1^Data Out 0;
						  .stSerial1.stComOut.D[1]  		:= TIIB[PCM A (EP6002-0002)]^COM RxPDO-Map Outputs Channel 1^Data Out 1;
						  .stSerial1.stComOut.D[2]  		:= TIIB[PCM A (EP6002-0002)]^COM RxPDO-Map Outputs Channel 1^Data Out 2;
						  .stSerial1.stComOut.D[3]  		:= TIIB[PCM A (EP6002-0002)]^COM RxPDO-Map Outputs Channel 1^Data Out 3;
						  .stSerial1.stComOut.D[4]  		:= TIIB[PCM A (EP6002-0002)]^COM RxPDO-Map Outputs Channel 1^Data Out 4;
						  .stSerial1.stComOut.D[5]  		:= TIIB[PCM A (EP6002-0002)]^COM RxPDO-Map Outputs Channel 1^Data Out 5;
						  .stSerial1.stComOut.D[6]  		:= TIIB[PCM A (EP6002-0002)]^COM RxPDO-Map Outputs Channel 1^Data Out 6;
						  .stSerial1.stComOut.D[7]  		:= TIIB[PCM A (EP6002-0002)]^COM RxPDO-Map Outputs Channel 1^Data Out 7;
						  .stSerial1.stComOut.D[8]  		:= TIIB[PCM A (EP6002-0002)]^COM RxPDO-Map Outputs Channel 1^Data Out 8;
						  .stSerial1.stComOut.D[9]  		:= TIIB[PCM A (EP6002-0002)]^COM RxPDO-Map Outputs Channel 1^Data Out 9;
						  .stSerial1.stComOut.D[10]  		:= TIIB[PCM A (EP6002-0002)]^COM RxPDO-Map Outputs Channel 1^Data Out 10;
						  .stSerial1.stComOut.D[11]  		:= TIIB[PCM A (EP6002-0002)]^COM RxPDO-Map Outputs Channel 1^Data Out 11;
						  .stSerial1.stComOut.D[12]  		:= TIIB[PCM A (EP6002-0002)]^COM RxPDO-Map Outputs Channel 1^Data Out 12;
						  .stSerial1.stComOut.D[13]  		:= TIIB[PCM A (EP6002-0002)]^COM RxPDO-Map Outputs Channel 1^Data Out 13;
						  .stSerial1.stComOut.D[14]  		:= TIIB[PCM A (EP6002-0002)]^COM RxPDO-Map Outputs Channel 1^Data Out 14;
						  .stSerial1.stComOut.D[15]  		:= TIIB[PCM A (EP6002-0002)]^COM RxPDO-Map Outputs Channel 1^Data Out 15;
						  .stSerial1.stComOut.D[16]  		:= TIIB[PCM A (EP6002-0002)]^COM RxPDO-Map Outputs Channel 1^Data Out 16;
						  .stSerial1.stComOut.D[17]  		:= TIIB[PCM A (EP6002-0002)]^COM RxPDO-Map Outputs Channel 1^Data Out 17;
						  .stSerial1.stComOut.D[18]  		:= TIIB[PCM A (EP6002-0002)]^COM RxPDO-Map Outputs Channel 1^Data Out 18;
						  .stSerial1.stComOut.D[19]  		:= TIIB[PCM A (EP6002-0002)]^COM RxPDO-Map Outputs Channel 1^Data Out 19;
						  .stSerial1.stComOut.D[20]  		:= TIIB[PCM A (EP6002-0002)]^COM RxPDO-Map Outputs Channel 1^Data Out 20;
						  .stSerial1.stComOut.D[21]  		:= TIIB[PCM A (EP6002-0002)]^COM RxPDO-Map Outputs Channel 1^Data Out 21;
						  
						  .stSerial2.stComOut.D[0]  		:= TIIB[PCM A (EP6002-0002)]^COM RxPDO-Map Outputs Channel 2^Data Out 0;
						  .stSerial2.stComOut.D[1]  		:= TIIB[PCM A (EP6002-0002)]^COM RxPDO-Map Outputs Channel 2^Data Out 1;
						  .stSerial2.stComOut.D[2]  		:= TIIB[PCM A (EP6002-0002)]^COM RxPDO-Map Outputs Channel 2^Data Out 2;
						  .stSerial2.stComOut.D[3]  		:= TIIB[PCM A (EP6002-0002)]^COM RxPDO-Map Outputs Channel 2^Data Out 3;
						  .stSerial2.stComOut.D[4]  		:= TIIB[PCM A (EP6002-0002)]^COM RxPDO-Map Outputs Channel 2^Data Out 4;
						  .stSerial2.stComOut.D[5]  		:= TIIB[PCM A (EP6002-0002)]^COM RxPDO-Map Outputs Channel 2^Data Out 5;
						  .stSerial2.stComOut.D[6]  		:= TIIB[PCM A (EP6002-0002)]^COM RxPDO-Map Outputs Channel 2^Data Out 6;
						  .stSerial2.stComOut.D[7]  		:= TIIB[PCM A (EP6002-0002)]^COM RxPDO-Map Outputs Channel 2^Data Out 7;
						  .stSerial2.stComOut.D[8]  		:= TIIB[PCM A (EP6002-0002)]^COM RxPDO-Map Outputs Channel 2^Data Out 8;
						  .stSerial2.stComOut.D[9]  		:= TIIB[PCM A (EP6002-0002)]^COM RxPDO-Map Outputs Channel 2^Data Out 9;
						  .stSerial2.stComOut.D[10] 	 	:= TIIB[PCM A (EP6002-0002)]^COM RxPDO-Map Outputs Channel 2^Data Out 10;
						  .stSerial2.stComOut.D[11] 	 	:= TIIB[PCM A (EP6002-0002)]^COM RxPDO-Map Outputs Channel 2^Data Out 11;
						  .stSerial2.stComOut.D[12] 	 	:= TIIB[PCM A (EP6002-0002)]^COM RxPDO-Map Outputs Channel 2^Data Out 12;
						  .stSerial2.stComOut.D[13] 	 	:= TIIB[PCM A (EP6002-0002)]^COM RxPDO-Map Outputs Channel 2^Data Out 13;
						  .stSerial2.stComOut.D[14] 	 	:= TIIB[PCM A (EP6002-0002)]^COM RxPDO-Map Outputs Channel 2^Data Out 14;
						  .stSerial2.stComOut.D[15] 	 	:= TIIB[PCM A (EP6002-0002)]^COM RxPDO-Map Outputs Channel 2^Data Out 15;
						  .stSerial2.stComOut.D[16] 	 	:= TIIB[PCM A (EP6002-0002)]^COM RxPDO-Map Outputs Channel 2^Data Out 16;
						  .stSerial2.stComOut.D[17] 	 	:= TIIB[PCM A (EP6002-0002)]^COM RxPDO-Map Outputs Channel 2^Data Out 17;
						  .stSerial2.stComOut.D[18] 	 	:= TIIB[PCM A (EP6002-0002)]^COM RxPDO-Map Outputs Channel 2^Data Out 18;
						  .stSerial2.stComOut.D[19] 	 	:= TIIB[PCM A (EP6002-0002)]^COM RxPDO-Map Outputs Channel 2^Data Out 19;
						  .stSerial2.stComOut.D[20] 	 	:= TIIB[PCM A (EP6002-0002)]^COM RxPDO-Map Outputs Channel 2^Data Out 20;
						  .stSerial2.stComOut.D[21] 	 	:= TIIB[PCM A (EP6002-0002)]^COM RxPDO-Map Outputs Channel 2^Data Out 21;
'}
PCMA : FB_PressureControlModule;

{attribute 'pytmc' := 'pv: XCS:SDS:PCM:B'}
{attribute 'TcLinkTo' := '.stPropAir1.i_iPressRB 	:= TIIB[PCM B (EP4374-0002)]^AI Inputs Channel 1^Value;
                          .stPropAir2.i_iPressRB 	:= TIIB[PCM B (EP4374-0002)]^AI Inputs Channel 2^Value;
                          .stPropAir1.q_iPressCt 	:= TIIB[PCM B (EP4374-0002)]^AO Outputs Channel 3^Analog output;
                          .stPropAir2.q_iPressCt 	:= TIIB[PCM B (EP4374-0002)]^AO Outputs Channel 4^Analog output;
                          .stSerial1.stComIn.Status := TIIB[PCM B (EP6002-0002)]^COM TxPDO-Map Inputs Channel 1^Status;
                          .stSerial2.stComIn.Status := TIIB[PCM B (EP6002-0002)]^COM TxPDO-Map Inputs Channel 2^Status;
                          .stSerial1.stComOut.Ctrl 	:= TIIB[PCM B (EP6002-0002)]^COM RxPDO-Map Outputs Channel 1^Ctrl;
                          .stSerial2.stComOut.Ctrl 	:= TIIB[PCM B (EP6002-0002)]^COM RxPDO-Map Outputs Channel 2^Ctrl;
                          .stBaseIO.i_SyncUnitWC 	:= TIIB[PCM B (EP1111)]^WcState^WcState;
'}
PCMB : FB_PressureControlModule;

{attribute 'pytmc' := 'pv: XCS:SDS:PCM:C'}
{attribute 'TcLinkTo' := '.stPropAir1.i_iPressRB 	:= TIIB[PCM C (EP4374-0002)]^AI Inputs Channel 1^Value;
                          .stPropAir2.i_iPressRB 	:= TIIB[PCM C (EP4374-0002)]^AI Inputs Channel 2^Value;
                          .stPropAir1.q_iPressCt 	:= TIIB[PCM C (EP4374-0002)]^AO Outputs Channel 3^Analog output;
                          .stPropAir2.q_iPressCt 	:= TIIB[PCM C (EP4374-0002)]^AO Outputs Channel 4^Analog output;
                          .stSerial1.stComIn.Status := TIIB[PCM C (EP6002-0002)]^COM TxPDO-Map Inputs Channel 1^Status;
                          .stSerial2.stComIn.Status := TIIB[PCM C (EP6002-0002)]^COM TxPDO-Map Inputs Channel 2^Status;
                          .stSerial1.stComOut.Ctrl 	:= TIIB[PCM C (EP6002-0002)]^COM RxPDO-Map Outputs Channel 1^Ctrl;
                          .stSerial2.stComOut.Ctrl 	:= TIIB[PCM C (EP6002-0002)]^COM RxPDO-Map Outputs Channel 2^Ctrl;
                          .stBaseIO.i_SyncUnitWC 	:= TIIB[PCM C (EP1111)]^WcState^WcState;
						  '}
PCMC : FB_PressureControlModule;

{attribute 'pytmc' := 'pv: XCS:SDS:PCM:D'}
{attribute 'TcLinkTo' := '.stPropAir1.i_iPressRB 	:= TIIB[PCM D (EP4374-0002)]^AI Inputs Channel 1^Value;
                          .stPropAir2.i_iPressRB 	:= TIIB[PCM D (EP4374-0002)]^AI Inputs Channel 2^Value;
                          .stPropAir1.q_iPressCt 	:= TIIB[PCM D (EP4374-0002)]^AO Outputs Channel 3^Analog output;
                          .stPropAir2.q_iPressCt 	:= TIIB[PCM D (EP4374-0002)]^AO Outputs Channel 4^Analog output;
                          .stSerial1.stComIn.Status := TIIB[PCM D (EP6002-0002)]^COM TxPDO-Map Inputs Channel 1^Status;
                          .stSerial2.stComIn.Status := TIIB[PCM D (EP6002-0002)]^COM TxPDO-Map Inputs Channel 2^Status;
                          .stSerial1.stComOut.Ctrl 	:= TIIB[PCM D (EP6002-0002)]^COM RxPDO-Map Outputs Channel 1^Ctrl;
                          .stSerial2.stComOut.Ctrl 	:= TIIB[PCM D (EP6002-0002)]^COM RxPDO-Map Outputs Channel 2^Ctrl;
                          .stBaseIO.i_SyncUnitWC 	:= TIIB[PCM D (EP1111)]^WcState^WcState;
						  '}
PCMD : FB_PressureControlModule;

{attribute 'pytmc' := 'pv: XCS:SDS:MAN'}
{attribute 'TcLinkTo' := '.stValve[1].qxDO := TIIB[Gas_Mani_ValveCtrl (EP2338-0001)]^Channel 9^Output;
                          .stValve[1].ixOPN := TIIB[Gas_Mani_ValveRbk (EP2338-0001)]^Channel 1^Input;
                          .stValve[2].qxDO := TIIB[Gas_Mani_ValveCtrl (EP2338-0001)]^Channel 10^Output;
                          .stValve[2].ixOPN := TIIB[Gas_Mani_ValveRbk (EP2338-0001)]^Channel 2^Input;
                          .stValve[3].qxDO := TIIB[Gas_Mani_ValveCtrl (EP2338-0001)]^Channel 11^Output;
                          .stValve[3].ixOPN := TIIB[Gas_Mani_ValveRbk (EP2338-0001)]^Channel 3^Input;
                          .stValve[4].qxDO := TIIB[Gas_Mani_ValveCtrl (EP2338-0001)]^Channel 12^Output;
                          .stValve[4].ixOPN := TIIB[Gas_Mani_ValveRbk (EP2338-0001)]^Channel 4^Input;
                          .stValve[5].qxDO := TIIB[Gas_Mani_ValveCtrl (EP2338-0001)]^Channel 13^Output;
                          .stValve[5].ixOPN := TIIB[Gas_Mani_ValveRbk (EP2338-0001)]^Channel 5^Input;
                          .stValve[6].qxDO := TIIB[Gas_Mani_ValveCtrl (EP2338-0001)]^Channel 14^Output;
                          .stValve[6].ixOPN := TIIB[Gas_Mani_ValveRbk (EP2338-0001)]^Channel 6^Input;
                          .stValve[7].qxDO := TIIB[Gas_Mani_ValveCtrl (EP2338-0001)]^Channel 15^Output;
                          .stValve[7].ixOPN := TIIB[Gas_Mani_ValveRbk (EP2338-0001)]^Channel 7^Input;
                          .stBaseIO.i_SyncUnitWC :=	TIID^MAIN (EtherCAT)^Gas_Mani (EP1111)^WcState^WcState;
'}
GasMan : FB_GasManifold;

{attribute 'pytmc' := 'pv: XCS:SDS:MFM:A'}
{attribute 'TcLinkTo' := '.stMFM.i_rFlow := TIID^MAIN (EtherCAT)^Bronkhorst MFM A^TxPDO Map^fMeasure;
                          .stMFM.q_rSetpoint := TIID^MAIN (EtherCAT)^Bronkhorst MFM A^RxPDO Map^fSetpoint;
'}
BronkhorstA : FB_BronkhorstMFM;

{attribute 'pytmc' := 'pv: XCS:SDS:MFM:B'}
{attribute 'TcLinkTo' := '.stMFM.i_rFlow 		:= TIIB[Bronkhorst MFM B]^TxPDO Map^fMeasure;
                          .stMFM.q_rSetpoint 	:=  TIIB[Bronkhorst MFM B]^RxPDO Map^fSetpoint;
'}
BronkhorstB : FB_BronkhorstMFM;

{attribute 'pytmc' := 'pv: XCS:SDS:MFM:C'}
{attribute 'TcLinkTo' := '.stMFM.i_rFlow := TIID^MAIN (EtherCAT)^Bronkhorst MFM C^TxPDO Map^fMeasure;
                          .stMFM.q_rSetpoint := TIID^MAIN (EtherCAT)^Bronkhorst MFM C^RxPDO Map^fSetpoint;
'}
BronkhorstC : FB_BronkhorstMFM;

{attribute 'pytmc' := 'pv: XCS:SDS:MFM:D'}
{attribute 'TcLinkTo' := '.stMFM.i_rFlow := TIID^MAIN (EtherCAT)^Bronkhorst MFM D^TxPDO Map^fMeasure;
                          .stMFM.q_rSetpoint := TIID^MAIN (EtherCAT)^Bronkhorst MFM D^RxPDO Map^fSetpoint;
'}
BronkhorstD : FB_BronkhorstMFM;

{attribute 'pytmc' := 'pv: XCS:SDS:SPR:A'}
{attribute 'TcLinkTo' := '.q_xDO1 := TIIB[Solenoid Pair A Digital IO (EP2338-0001)]^Channel 9^Output;
                          .q_xDO2 := TIIB[Solenoid Pair A Digital IO (EP2338-0001)]^Channel 10^Output;
'}
SolenoidPairA : FB_SolenoidPair;


END_VAR

// ---- POUs/MAIN.TcPOU
PROGRAM MAIN
VAR

END_VAR

M3SelectorA();
M3SelectorB();
M3SelectorC();
M3SelectorD();
PCMA();
PCMB();
PCMC();
PCMD();
GasMan();
BronkhorstA();
BronkhorstB();
BronkhorstC();
BronkhorstD();
SolenoidPairA();

(* Following execution of all the programs, set the first pass false *)
g_xFirstPass := FALSE;

END_PROGRAM
